# B&R Automation Studio project vibratorControlWithCurrentController (part 7)

#### Variables.var - Local variables
```iecst
VAR CONSTANT
	CYCLE_TIME_us : REAL := 1600.0;
	CYCLE_TIME_s : REAL := 0.0016;
	PI : REAL := 3.1415926536;
END_VAR
VAR
	acc : acc_typ;
	i : USINT;
	vibratorControl_0 : ARRAY[0..NUM_VIBRATOR] OF vibratorControl := [2((startPercentBoost:=5))];
	local : ARRAY[0..NUM_VIBRATOR] OF local_typ;
	MTFilterMovingAverage_0 : ARRAY[0..NUM_VIBRATOR] OF MTFilterMovingAverage;
	MTBasicsTimeDelay_0 : ARRAY[0..NUM_VIBRATOR] OF MTBasicsTimeDelay;
	GetPhaseDifference_0 : ARRAY[0..NUM_VIBRATOR] OF GetPhaseDifference;
	hmiAccelerometerPercent : REAL;
END_VAR
```

#### LocalFunctions.fun
```iecst
{REDUND_ERROR} FUNCTION_BLOCK vibratorControl (*TODO: Add your comment here*) (*$GROUP=User,$CAT=User,$GROUPICON=User.png,$CATICON=User.png*)
	VAR_INPUT
		enable : BOOL;
		amplitude : REAL;
		percent : REAL;
		vibratorType : USINT;
		machineType : USINT;
		manualFrequency : REAL;
		manualControl : BOOL;
		linearizationAmplitude : ARRAY[0..4] OF REAL;
		linearizationFrequencies : ARRAY[0..4] OF REAL;
		pAxis : UDINT;
		manualBrake : BOOL;
		boostVelocityLow : REAL := 180;
		boostVelocityHigh : REAL;
		brakeVelocity : REAL;
		boostFrequency : REAL;
		brakeFrequency : REAL;
		boostAmplitude : REAL;
		brakeAmplitude : REAL;
		manualBoost : BOOL;
		currAccelerometerValue : REAL;
		currAccelerometerPercent : REAL;
		manualBrakeTime : REAL;
		manualBrakeAmplitudeEnd : REAL;
		manualBrakeFrequencyEnd : REAL;
		activateMinMax : BOOL;
		disableBoost : BOOL;
	END_VAR
	VAR_OUTPUT
		frequency_out : REAL;
		amplitude_out : REAL;
		phaseShift : REAL := 0;
		sin_out : REAL;
		accelerationStart : REAL;
		minAcceleration : REAL;
		minAccelerationTime : REAL;
		caliBoostVelocityLow : REAL;
		caliBoostVelocityHigh : REAL;
		estimatedPercent : REAL;
		minBreakPercent : REAL;
		maxBoostPercent : REAL;
		filteredAccelerometerPercent : REAL;
	END_VAR
	VAR
		state : UINT;
		oldPercent : REAL;
		phi : REAL;
		sine : REAL;
		time : REAL;
		oldMachineType : USINT := 222; (*222 to make sure gets initialized*)
		addBrakeAmplitude : REAL;
		enableBrake : BOOL := TRUE;
		phaseShiftLocal : REAL;
		minBrakeTime : REAL := 0;
		j : UINT;
		MTLookUpTable_0 : MTLookUpTable;
		frequency : REAL;
		MC_BR_CyclicWrite_0 : MC_BR_CyclicWrite;
		old_sin : REAL;
		sin_ref : REAL;
		startPercentBoost : REAL;
		sin_abs : REAL;
		oldVibratorType : USINT;
		brakeStartDelay : REAL;
		brakePercent : REAL;
		timeStart : REAL;
		accelerationStart20pct : REAL;
		MTDataMinMax_0 : MTDataMinMax;
		MTFilterMovingAverage_0 : MTFilterMovingAverage;
		oldCurrAccelerometerValue : REAL;
		boostHighLowSeperatorPercent : REAL := 50.0;
	END_VAR
END_FUNCTION_BLOCK

FUNCTION getPercentFromAcceleration : REAL
	VAR_INPUT
		acc : REAL;
		vibratorType : USINT; (*0=CF, 1=LF*)
		machineType : USINT; (*0=small, 1=big*)
	END_VAR
END_FUNCTION

FUNCTION getAccelerationFromPercent : REAL
	VAR_INPUT
		percent : REAL;
		vibratorType : USINT; (*0=CF, 1=LF*)
		machineType : USINT; (*0=small, 1=big*)
	END_VAR
END_FUNCTION

FUNCTION applyBrake : REAL
	VAR_INPUT
		percent : REAL;
		brakeVelocity : REAL; (*accValue/s*)
		vibratorType : USINT; (*0=CF, 1=LF*)
		machineType : USINT; (*0=small, 1=big*)
	END_VAR
	VAR
		acc : REAL;
		bigBowlChange : REAL := 48000;
	END_VAR
END_FUNCTION

FUNCTION applyBoost : REAL
	VAR_INPUT
		percent : REAL;
		boostVelocity : REAL; (*accValue/s*)
		vibratorType : USINT; (*0=CF, 1=LF*)
		machineType : USINT; (*0=small, 1=big*)
	END_VAR
	VAR
		acc : REAL;
	END_VAR
END_FUNCTION

FUNCTION_BLOCK GetPhaseDifference
	VAR_INPUT
		Enable : BOOL;
		ReferenceSignal : REAL;
		Signal : REAL;
	END_VAR
	VAR_OUTPUT
		Phase : REAL;
		PhaseInv : REAL;
	END_VAR
	VAR
		x : ARRAY[0..MAX_SIGNAL_LENGTH] OF REAL;
		y : ARRAY[0..MAX_SIGNAL_LENGTH] OF REAL;
		r : ARRAY[0..MAX_OUTPUT_LENGTH] OF REAL;
	END_VAR
	VAR CONSTANT
		MAX_SIGNAL_LENGTH : UINT := 19;
		MAX_OUTPUT_LENGTH : UINT := (MAX_SIGNAL_LENGTH*2)+1;
	END_VAR
	VAR
		i : {REDUND_UNREPLICABLE} UINT;
		sum : {REDUND_UNREPLICABLE} REAL;
		offset : {REDUND_UNREPLICABLE} INT;
		j : {REDUND_UNREPLICABLE} UINT;
		maxVal : {REDUND_UNREPLICABLE} REAL;
		maxIdx : {REDUND_UNREPLICABLE} UINT;
		state : UINT;
		idx : UINT;
		minVal : REAL;
		minIdx : UINT;
	END_VAR
END_FUNCTION_BLOCK
```

#### LocalFunctions.st
```iecst
FUNCTION_BLOCK vibratorControl

	CASE state OF

		0:
			IF enable THEN
				IF vibratorType=0 THEN
					state := 5;
				ELSE
					//LF
					state := 8;
				END_IF
			END_IF

		5: // CF Running
			IF manualControl THEN
				state := 200;
			ELSIF percent < estimatedPercent AND frequency <> 0.0 THEN
				time := 0;
				brakePercent := percent;
				state := 20;
			ELSIF percent > estimatedPercent AND frequency <> 0.0 THEN
				time := 0;
				oldPercent := percent;
				state := 10;
			ELSE
				amplitude_out := amplitude;
				MTLookUpTable_0.InX := amplitude;
				MTLookUpTable_0();
				frequency := MTLookUpTable_0.Out;
			END_IF

		8: // LF Running
			IF manualControl THEN
				state := 200;
			ELSE
				amplitude_out := amplitude;
				MTLookUpTable_0.InX := amplitude;
				MTLookUpTable_0();
				frequency := MTLookUpTable_0.Out;
			END_IF

		10: // wait for zero crossing
			IF sin_ref >= 0.0 AND old_sin < 0.0 THEN
				amplitude_out := boostAmplitude;
				estimatedPercent := MAX(estimatedPercent, startPercentBoost);

				MTDataMinMax_0.Enable := FALSE;
				MTDataMinMax_0();
				state := 15;
			ELSIF sin_ref <= 0.0 AND old_sin > 0.0 THEN
				amplitude_out := boostAmplitude;
				estimatedPercent := MAX(estimatedPercent, startPercentBoost);

				MTDataMinMax_0.Enable := FALSE;
				MTDataMinMax_0();
				state := 15;
			END_IF

		15: // Boosting
			amplitude_out := boostAmplitude;
			frequency := boostFrequency;

			IF estimatedPercent <= boostHighLowSeperatorPercent THEN
				estimatedPercent := applyBoost(estimatedPercent, boostVelocityLow, vibratorType, machineType);
			ELSE
				estimatedPercent := applyBoost(estimatedPercent, boostVelocityHigh, vibratorType, machineType);
			END_IF
			time := time + CYCLE_TIME_s;

			IF percent <> oldPercent THEN
				state := 5;
			ELSIF estimatedPercent >= percent OR disableBoost THEN
				estimatedPercent := percent;
				state := 5;
			END_IF

		20:
			IF sin_ref >= 0.0 AND old_sin < 0.0 THEN
				amplitude_out := brakeAmplitude;
				phi := phi - (PI/2.0);

				MTDataMinMax_0.Enable := FALSE;
				MTDataMinMax_0();
				state := 25;
			ELSIF sin_ref <= 0.0 AND old_sin > 0.0 THEN
				amplitude_out := brakeAmplitude;
				phi := phi - (PI/2.0);

				MTDataMinMax_0.Enable := FALSE;
				MTDataMinMax_0();
				state := 25;
			END_IF

		25: // Braking
			amplitude_out := brakeAmplitude;
			frequency := brakeFrequency;

			estimatedPercent := applyBrake(estimatedPercent, brakeVelocity, vibratorType, machineType);

			time := time + CYCLE_TIME_s;

			IF estimatedPercent <= brakePercent THEN
				estimatedPercent := brakePercent;

				amplitude_out := 0.0;
				phi := phi + (PI/2.0);
				state := 5;
			END_IF

		100:
			amplitude_out := amplitude;
			MTLookUpTable_0.InX := amplitude;
			MTLookUpTable_0();
			frequency := MTLookUpTable_0.Out;

		200:
			frequency := manualFrequency;
			amplitude_out := amplitude;

			IF manualBrake THEN
				state := 210;
				time := 0;
			ELSIF manualBoost THEN
				time := 0.0;
				state := 250;
			ELSIF NOT manualControl THEN
				estimatedPercent := 0;
				MTLookUpTable_0.Enable := FALSE;
				MTLookUpTable_0();
				state := 5;
			END_IF

		210:
			IF sin_ref >= 0.0 AND old_sin < 0.0 THEN
				amplitude_out := brakeAmplitude;
				phi := phi - (PI/2.0);
				accelerationStart := currAccelerometerValue;
				minAcceleration := 99999999;
				state := 220;
			ELSIF sin_ref <= 0.0 AND old_sin > 0.0 THEN
				amplitude_out := brakeAmplitude;
				phi := phi - (PI/2.0);
				accelerationStart := currAccelerometerValue;
				timeStart := 0;
				minAcceleration := 99999999;
				state := 220;
			END_IF

		220: // Braking
			amplitude_out := brakeAmplitude;
			frequency := brakeFrequency;

			time := time + CYCLE_TIME_s;

			IF time > manualBrakeTime OR NOT manualBrake THEN
				amplitude_out := manualBrakeAmplitudeEnd;
				frequency := manualBrakeFrequencyEnd;
				phi := phi + (PI/2.0);
				state := 230;
			END_IF

			IF currAccelerometerValue < minAcceleration THEN
				IF timeStart > 0 AND time-timeStart >= CYCLE_TIME_s*2 THEN
					accelerationStart := accelerationStart20pct;
					minAcceleration := currAccelerometerValue;
					minAccelerationTime := time-timeStart;
				ELSE
					minAcceleration := currAccelerometerValue;
					minAccelerationTime := time;
				END_IF
			END_IF

			// If acceleromter falls more than 20% save that point as "start point".
			IF currAccelerometerValue < (accelerationStart*0.8) AND timeStart=0 THEN
				accelerationStart20pct := currAccelerometerValue;
				timeStart := time;
			END_IF

		230:
			IF currAccelerometerValue < minAcceleration THEN
				IF timeStart > 0 AND time-timeStart >= CYCLE_TIME_s*2 THEN
					accelerationStart := accelerationStart20pct;
					minAcceleration := currAccelerometerValue;
					minAccelerationTime := time-timeStart;
				ELSE
					minAcceleration := currAccelerometerValue;
					minAccelerationTime := time;
				END_IF
			END_IF

			// If acceleromter falls more than 20% save that point as "start point".
			IF currAccelerometerValue < (accelerationStart*0.8) AND timeStart=0 THEN
				accelerationStart20pct := currAccelerometerValue;
				timeStart := time;
			END_IF

			IF NOT manualBrake THEN
				amplitude_out := 0;
				state := 200;
			END_IF

		250: // wait for zero crossing
			IF sin_ref >= 0.0 AND old_sin < 0.0 THEN
				amplitude_out := boostAmplitude;
				state := 260;
			ELSIF sin_ref <= 0.0 AND old_sin > 0.0 THEN
				amplitude_out := boostAmplitude;
				state := 260;
			END_IF

		260: // Boosting
			amplitude_out := boostAmplitude;
			frequency := boostFrequency;

			time := time + CYCLE_TIME_s;
			caliBoostVelocityLow := currAccelerometerValue / time;

			IF time >= 0.5 OR NOT manualBoost OR currAccelerometerPercent >= 50.0 THEN
				time := 0;
				accelerationStart := currAccelerometerValue;
				state := 270;
			END_IF

		270:
			amplitude_out := boostAmplitude;
			frequency := boostFrequency;

			time := time + CYCLE_TIME_s;
			caliBoostVelocityHigh := (currAccelerometerValue-accelerationStart) / time;

			IF time >= 0.5 THEN
				caliBoostVelocityHigh := caliBoostVelocityLow;

				amplitude_out := 0.0;
				state := 280;
			ELSIF NOT manualBoost OR currAccelerometerPercent >= 90.0 THEN
				amplitude_out := 0.0;
				state := 280;
			END_IF

		280:
			IF NOT manualBoost THEN
				state := 200;
			END_IF

	END_CASE

	IF NOT enable AND state <> 0 THEN
		estimatedPercent := 0;
		state := 0;
		amplitude_out := 0;
		frequency_out := 0;
	END_IF

	// Lookup table for frequencies
	IF enable AND NOT MTLookUpTable_0.Enable THEN
		MTLookUpTable_0.Mode := mtLOOKUP_LINEAR_EXTRAPOLATION;

		MTLookUpTable_0.NumberOfNodes := 0;
		FOR j:=0 TO 4 DO
			IF linearizationAmplitude[j]=0.0 THEN
				EXIT;
			END_IF
			MTLookUpTable_0.NodeVectorX[j] := linearizationAmplitude[j];
			MTLookUpTable_0.FcnValues[j] := linearizationFrequencies[j];
			MTLookUpTable_0.NumberOfNodes := MTLookUpTable_0.NumberOfNodes + 1;
		END_FOR
	END_IF
	MTLookUpTable_0.Enable := enable;
	MTLookUpTable_0();

	IF activateMinMax OR manualControl THEN
		IF currAccelerometerValue <> oldCurrAccelerometerValue THEN
			oldCurrAccelerometerValue := currAccelerometerValue;

			MTFilterMovingAverage_0.Enable := TRUE;
			MTFilterMovingAverage_0.In := currAccelerometerValue;
			MTFilterMovingAverage_0.WindowLength := 10;
			MTFilterMovingAverage_0();

			MTDataMinMax_0.Enable := TRUE;
			MTDataMinMax_0.In := MTFilterMovingAverage_0.Out;
			MTDataMinMax_0();
			minBreakPercent := getPercentFromAcceleration(MTDataMinMax_0.MinValue ,vibratorType,machineType);
			maxBoostPercent := getPercentFromAcceleration(MTDataMinMax_0.MaxValue ,vibratorType,machineType);
			filteredAccelerometerPercent := getPercentFromAcceleration(MTFilterMovingAverage_0.Out,vibratorType,machineType);
		END_IF
	END_IF

	old_sin := sin_ref;

	// create sinewave amplitude with defined frequency
	sin_out := amplitude_out*SIN(phi+phaseShift);
	sin_abs := ABS(sin_out);
	phi := fmod(phi + frequency*2*PI*CYCLE_TIME_s, 2*PI);
	sin_ref := SIN(phi+phaseShift);
	phaseShift := fmod(phaseShift, 2*PI);
	phaseShiftLocal := fmod(phaseShiftLocal, 2*PI);

	// Write sine wave to vibrator parID
	MC_BR_CyclicWrite_0.Enable := enable;
	MC_BR_CyclicWrite_0.Axis := pAxis;
	MC_BR_CyclicWrite_0.DataType := ncPAR_TYP_REAL;
	MC_BR_CyclicWrite_0.DataAddress := ADR(sin_out);
	MC_BR_CyclicWrite_0.ParID := ACP10PAR_USER_R4_VAR1;
	MC_BR_CyclicWrite_0();

	// If machineType changes we must change parameters.
	IF machineType <> oldMachineType OR vibratorType <> oldVibratorType THEN
		oldMachineType := machineType;
		oldVibratorType := vibratorType;

		IF machineType=0 THEN
			IF vibratorType=0 THEN
				// small CF
			//	startPercentBoost := 5.0;
				brakeAmplitude := 1.5;
				boostAmplitude := 1.5;
				boostVelocityLow := 60500;
			ELSE
				// small LF
			//	startPercentBoost := 10.0;
				brakeAmplitude := 0.06;
				boostAmplitude := 0.12;
				boostVelocityLow := 29195;
			END_IF
		ELSE
			IF vibratorType=0 THEN
				// big CF
			//	startPercentBoost := 5.0;
				brakeAmplitude := 2.5;
				boostAmplitude := 2.5;
				boostVelocityLow := 29195;
			ELSE
				// big LF
			//	startPercentBoost := 10.0;
				brakeAmplitude := 0.06;
				boostAmplitude := 0.12;
				boostVelocityLow := 29195;
			END_IF
		END_IF

	END_IF

END_FUNCTION_BLOCK

FUNCTION getPercentFromAcceleration

	IF machineType=0 THEN
		IF vibratorType=0 THEN
			// 10%=2756 , 100%=17420
			getPercentFromAcceleration := (acc-1126.7)/162.93;
		ELSE
			// 10%=1300 , 100%=10140
			getPercentFromAcceleration := (acc-317.78)/98.222;
		END_IF
	ELSE
		IF vibratorType=0 THEN
			// 10%=1456 , 100%=8060
			getPercentFromAcceleration := (acc-722.22)/73.378;;
		ELSE
			// 10%=1508 , 100%=8840
			getPercentFromAcceleration := (acc-693.33)/81.467;
		END_IF
	END_IF

END_FUNCTION

FUNCTION getAccelerationFromPercent

	IF machineType=0 THEN
		IF vibratorType=0 THEN
			// 10%=2756 , 100%=17420
			getAccelerationFromPercent := percent*162.93+1126.7;
		ELSE
			// 10%=1300 , 100%=10140
			getAccelerationFromPercent := percent*98.222+317.78;
		END_IF
	ELSE
		IF vibratorType=0 THEN
			// 10%=1456 , 100%=8060
			getAccelerationFromPercent := percent*73.378+722.22;
		ELSE
			// 10%=1508 , 100%=8840
			getAccelerationFromPercent := percent*81.467+693.33;
		END_IF
	END_IF

END_FUNCTION

FUNCTION applyBoost
	acc := getAccelerationFromPercent(percent,vibratorType,machineType);
	applyBoost := getPercentFromAcceleration(acc+(boostVelocity*CYCLE_TIME_s),vibratorType,machineType);

//	IF machineType=0 THEN
//		IF vibratorType=0 THEN
//			applyBoost := getPercentFromAcceleration(acc+(55910*CYCLE_TIME_s),vibratorType,machineType);
//		ELSE
//			applyBoost := getPercentFromAcceleration(acc+(29195*CYCLE_TIME_s),vibratorType,machineType);
//		END_IF
//	ELSE
//		IF vibratorType=0 THEN
//			// big CF
//			applyBoost := getPercentFromAcceleration(acc+(29195*CYCLE_TIME_s),vibratorType,machineType);
//		ELSE
//			applyBoost := getPercentFromAcceleration(acc+(29195*CYCLE_TIME_s),vibratorType,machineType);
//		END_IF
//	END_IF

END_FUNCTION

FUNCTION applyBrake
	acc := getAccelerationFromPercent(percent,vibratorType,machineType);
	applyBrake := getPercentFromAcceleration(acc-(brakeVelocity*CYCLE_TIME_s),vibratorType,machineType);

	//	IF vibratorSize=0 THEN
	//		IF vibratorType=0 THEN
	//			applyBrake := getPercentFromAcceleration(acc-(48000*CYCLE_TIME_s),vibratorType,vibratorSize); //applyBrake := getPercentFromAcceleration(acc-(94349*CYCLE_TIME_s),vibratorType,vibratorSize);
	//		ELSE
	//			applyBrake := getPercentFromAcceleration(acc-(48000*CYCLE_TIME_s),vibratorType,vibratorSize);
	//		END_IF
	//	ELSE
	//		IF vibratorType=0 THEN
	//			// big CF
	//			applyBrake := getPercentFromAcceleration(acc-(42000*CYCLE_TIME_s),vibratorType,vibratorSize);
	//		ELSE
	//			applyBrake := getPercentFromAcceleration(acc-(48000*CYCLE_TIME_s),vibratorType,vibratorSize);
	//		END_IF
	//	END_IF

END_FUNCTION

FUNCTION_BLOCK GetPhaseDifference

	CASE state OF
		0:
			IF Enable THEN
				idx := 0;
				state := 10;
			END_IF

		10:
			x[idx] := ReferenceSignal;
			y[idx] := Signal;

			idx := idx + 1;

			IF idx > MAX_SIGNAL_LENGTH THEN
				idx := 0;
				state := 20;
			END_IF

		20:
			maxVal := 0;
			maxIdx := 0;
			minVal := 999999999;
			minIdx := 0;

			FOR i:=0 TO MAX_OUTPUT_LENGTH DO
				sum := 0;
				offset := UINT_TO_INT(i)-UINT_TO_INT(MAX_SIGNAL_LENGTH);
				FOR j:=0 TO MAX_SIGNAL_LENGTH DO
					IF UINT_TO_INT(j)+offset >= 0 AND UINT_TO_INT(j)+offset <= MAX_SIGNAL_LENGTH THEN
						sum := sum + (x[j] * y[j+offset]);
					END_IF
				END_FOR
				IF sum >= maxVal THEN
					maxVal := sum;
					maxIdx := i;
				END_IF
				IF sum <= minVal THEN
					minVal := sum;
					minIdx := i;
				END_IF

				r[i] := sum;
			END_FOR

			Phase := UINT_TO_REAL(maxIdx)-UINT_TO_REAL(MAX_SIGNAL_LENGTH);
			PhaseInv := UINT_TO_REAL(minIdx)-UINT_TO_REAL(MAX_SIGNAL_LENGTH);

			state := 10;

	END_CASE

	IF NOT Enable AND state > 0 THEN
		state := 0;
	END_IF

END_FUNCTION_BLOCK
```

### Program Logical/modules/main/vibrator/VibratorControl (IEC)

#### local.st - Init, cyclic, exit code
```iecst
PROGRAM _INIT

	FOR i:=0 TO NUM_VIBRATOR DO
		this ACCESS ADR(localVariables[i]);
		config ACCESS ADR(localVariables[i].config);

		// gets the task name and setup names for config and receipe types
		ST_name(0,ADR(this.configName),0);
		brdkStrCat(ADR(this.configName),ADR(':localVariables['));
		brdkStrAppendUdintToA(i,ADR(this.configName),0,-1);
		brdkStrCat(ADR(this.configName),ADR('].config'));

		this.VibFeedback_0.VibratorType := i;
		this.VibControl_0.VibratorType := i; // i=0=CF , i=1=LF
		this.Accelerometer_0.VibratorType := i; // i=0=CF , i=1=LF
		this.MpRecipeRegPar_Config.Enable := TRUE;
		config.emptyPercent := SEL(i=0,110,50);
		gVibratorInterface[i].cmd.emptyPercent := config.emptyPercent;
	END_FOR

END_PROGRAM

PROGRAM _CYCLIC

	FOR i:=0 TO NUM_VIBRATOR DO
		this ACCESS ADR(localVariables[i]);
		config ACCESS ADR(localVariables[i].config);
		hmi ACCESS ADR(localHmi[i]);

		modules;
	END_FOR

	// Watch Idx
	i := LIMIT(0, watchIdx, NUM_VIBRATOR);
	this ACCESS ADR(localVariables[i]);
	hmi ACCESS ADR(localHmi[i]);
	config ACCESS ADR(localVariables[i].config);

END_PROGRAM

PROGRAM _EXIT

END_PROGRAM
```

#### modules.st
```iecst
ACTION modules:

	// Function block for accelerometer processing
	this.Accelerometer_0.Enable := this.Accelerometer_0.ModuleOkCalibrationTool OR this.Accelerometer_0.ModuleOkBusCtrl;
	this.Accelerometer_0();

	// Function block for calculating airgap phase and amplitude
	this.VibFeedback_0.Enable := gVibratorInterface[i].status.powered;
	this.VibFeedback_0.Axis := SEL(i=0, ADR(gAxisVibL), ADR(gAxisVibC));
	this.VibFeedback_0.Amplitude_out := this.VibControl_0.amplitude_out;
	this.VibFeedback_0.Frequency := this.VibControl_0.frequency_out;
	this.VibFeedback_0.HoldPhase := this.VibControl_0.HoldPhase;
	this.VibFeedback_0.SinePhase := this.VibControl_0.SinePhase;
	this.VibFeedback_0.SineOut := this.VibControl_0.SineOut;
	this.VibFeedback_0.Braking := this.VibControl_0.Braking;
	this.VibFeedback_0.RawVib := this.Accelerometer_0.Raw; // only for phase verification
	this.VibFeedback_0.BrakingToAmplitudePct := this.VibControl_0.BrakingToAmplitudePct;
	this.VibFeedback_0();

	// Function block for closed loop phase and amplitude control, as well as setpoint generation for current controller
	this.VibControl_0.Enable := gVibratorInterface[i].status.powered;
	this.VibControl_0.Axis := SEL(i=0, ADR(gAxisVibL), ADR(gAxisVibC));
	this.VibControl_0.Percent := this.Accelerometer_0.Percent;
	this.VibControl_0.SetAmplitude := gVibratorInterface[i].status.percent;
	this.VibControl_0.ActPhase := this.VibFeedback_0.Phase;
	this.VibControl_0.ActPhaseValid := this.VibFeedback_0.PhaseValid;
	this.VibControl_0.ActPhaseAcc := this.VibFeedback_0.PhaseAcc;
	this.VibControl_0.ActAmplitude := SEL(this.testAccFeedback,this.VibFeedback_0.Amplitude,this.Accelerometer_0.Percent);
	this.VibControl_0.ActAmplitudeValid := this.VibFeedback_0.AmplitudeValid;
	this.VibControl_0.ManualControl := (gVibratorInterface[i].status.forcing) AND NOT gVibratorInterface[i].status.caliProdTest;
//	this.VibControl_0.AccPercent := this.Accelerometer_0.Percent;
	this.VibControl_0();
	hmi.frequencyTimes2 := this.VibControl_0.frequency_out*2.0; // to show on HMI

	// Config handling (it takes too much CPU to run in 0.8ms so we run it with a timer):
	this.timeConfig := this.timeConfig + CYCLE_TIME_us;
	IF this.timeConfig > 80000 THEN // 80ms
		this.timeConfig := 0;

		// Slow inputs every 80ms
		this.VibControl_0.config := ADR(config);
		this.VibFeedback_0.config := ADR(config);
		this.VibFeedback_0.UpdateFilter := this.VibControl_0.UpdateFilter;
		this.VibFeedback_0.Calibrating := gVibratorInterface[i].status.calibratingMode AND NOT this.VibControl_0.TestPulses;
		this.Accelerometer_0.MachineSize := config.MachineSize;
		this.VibFeedback_0.MachineSize := config.MachineSize;
		this.VibControl_0.MachineSize := config.MachineSize;
		this.VibControl_0.Calibrate := gVibratorInterface[i].status.calibratingMode;
		this.VibControl_0.RampUp := SEL(gVibratorInterface[i].status.rampUp > 0,0,100/(INT_TO_REAL(gVibratorInterface[i].status.rampUp)/1000)); // ms it takes to go from 0% to 100% -> 100ms ex. 100/0.1 = 1000%/s
		this.VibControl_0.ManualPercent := SEL(gVibratorInterface[i].parameter.speedPctManualTest > 0,this.VibControl_0.ManualPercent,gVibratorInterface[i].parameter.speedPctManualTest);
		this.VibControl_0.MinTimeInCount := config.minTimeInCount;
		this.VibControl_0.MinTimeInCountBigCf := config.minTimeInCountBigCf;

		// Slow outputs every 80ms
		gVibratorInterface[i].cmd.calibrationDone := this.VibControl_0.CalibrateDone;
		gVibratorInterface[i].cmd.testPulses := this.VibControl_0.TestPulses;
		gVibratorInterface[i].cmd.emptyPercent := config.emptyPercent;
		gVibratorInterface[i].parameter.machineSize := localVariables[0].config.MachineSize;
		this.VibControl_0.UpdateFilterDone := this.VibFeedback_0.UpdateFilterDone;
		localVariables[1].config.MachineSize := localVariables[0].config.MachineSize;
		hmi.calibrationNotActive := NOT this.VibControl_0.Calibrate;

		IF config.calibrationDone THEN
			config.timeInCalibrationSeconds := config.timeInCalibrationSeconds + 0.08; // Previously used PLC TIME but that gets destroyed by NTP. Rather use a counter even though it can't count if power is OFF.
			hmi.daysSinceCalibration := config.timeInCalibrationSeconds/86400; // Convert seconds to days.

			// Auto save every 30min
			timeElapsedMillis := timeElapsedMillis + 80;
			IF timeElapsedMillis > 1800000 THEN
				timeElapsedMillis := 0;
				this.SaveConfig := TRUE;
			END_IF

			// Only show this when calibration is done. Otherwise it will show 2 different numbers doing calibration which may confuse
			config.ressonanceFrequencyAt45Pct := config.maxFrequencySweep*2.0; // ressonance (mechanical) frequency is really 2 times output frequency.
		ELSE
			hmi.daysSinceCalibration := 99999;
		END_IF

		// Set max current depending which machine size.
		IF config.MachineSize=0 THEN
			this.VibControl_0.MaxCurr := SEL(i=0, 0.20, 2.0);
		ELSE
			this.VibControl_0.MaxCurr := SEL(i=0, 0.20, 3.1);
		END_IF

		// Set max current depending which machine size.
		IF config.MachineSize=0 THEN
			// Small bowl						  LF    CF
			hmi.minResonanceFrequency := SEL(i=0, 96, 96);
			hmi.maxResonanceFrequency := SEL(i=0, 106, 102);
			hmi.minCurrent := SEL(i=0, 0.04, 0.4);
			hmi.maxCurrent := SEL(i=0, 0.13, 1.3);
		ELSE
			// Big bowl							  LF    CF
			hmi.minResonanceFrequency := SEL(i=0, 96, 47);
			hmi.maxResonanceFrequency := SEL(i=0, 106, 52);
			hmi.minCurrent := SEL(i=0, 0.04, 0.4);
			hmi.maxCurrent := SEL(i=0, 0.13, 1.9);
		END_IF
		hmi.resonanceFrequencyOK := this.config.ressonanceFrequencyAt45Pct >= hmi.minResonanceFrequency AND this.config.ressonanceFrequencyAt45Pct <= hmi.maxResonanceFrequency;
		hmi.currentOK := this.config.maxCurrentUsed >= hmi.minCurrent AND this.config.maxCurrentUsed <= hmi.maxCurrent;

		// Interface calibration results to FAT (send if calibrate is stopped)
		IF this.VibControl_0.SendCaliResultToFAT THEN
			this.VibControl_0.SendCaliResultToFAT := FALSE;

			gVibratorInterface[i].status.calibrationResultFrequencyOK := hmi.resonanceFrequencyOK;
			gVibratorInterface[i].status.calibrationResultCurrentOK := hmi.currentOK;
			gVibratorInterface[i].status.calibrationResultFrequency := this.config.ressonanceFrequencyAt45Pct;
			gVibratorInterface[i].status.calibrationResultCurrent := this.config.maxCurrentUsed;
			gVibratorInterface[i].status.calibrationResultsReady := TRUE;
		END_IF
		gVibratorInterface[i].status.calibrationDone := config.calibrationDone;

		// set machinesize (cmd from FAT)
		IF gVibratorInterface[i].cmd.setCfType THEN
			gVibratorInterface[i].cmd.setCfType := FALSE;
			config.MachineSize := gVibratorInterface[i].parameter.CFType; //0=small , 1=big
			this.SaveConfig := TRUE;
		END_IF

		// State Machine to save config.
		CASE this.stateSave OF

			0:
				IF this.VibControl_0.SaveConfig AND gConfig.status.loaded THEN
					// Save from calibration
					gConfig.cmd.save := TRUE;
					gMachineInterface.cmd.requestSaveToT50 := TRUE;
					this.stateSave := 10;
				ELSIF this.SaveConfig AND gConfig.status.loaded THEN
					// Save because HMI variable changed.
					this.SaveConfig := FALSE;
					gConfig.cmd.save := TRUE;
					this.stateSave := 30;
				END_IF

			10:
				IF NOT gConfig.cmd.save THEN
					this.VibControl_0.SaveConfigDone := TRUE;
					this.stateSave := 20;
				END_IF

			20:
				IF NOT this.VibControl_0.SaveConfig THEN
					this.VibControl_0.SaveConfigDone := FALSE;
					this.stateSave := 0;
				END_IF

			30:
				IF NOT gConfig.cmd.save THEN
					this.stateSave := 0;
				END_IF

		END_CASE

	this.MpRecipeRegPar_Config(MpLink := ADR(mpRecipe), PVName := ADR(this.configName), Category := ADR('config'));
END_IF

END_ACTION
```

#### Types.typ - Local data types
```iecst
TYPE
	hmi_typ : 	STRUCT
		NeedCalibration : BOOL;
		CalibrationStatus : calibrationResult_enum;
		daysSinceCalibration : REAL := 99999;
		calibrationNotActive : BOOL;
		resonanceFrequencyOK : BOOL;
		currentOK : BOOL;
		minCurrent : REAL;
		maxCurrent : REAL;
		minResonanceFrequency : REAL;
		maxResonanceFrequency : REAL;
		frequencyTimes2 : REAL;
	END_STRUCT;
	local_typ : 	STRUCT
		VibFeedback_0 : VibFeedback;
		VibControl_0 : VibControl;
		Accelerometer_0 : Accelerometer;
		useAccPhase : BOOL;
		MpRecipeRegPar_Config : MpRecipeRegPar;
		VibFeedback_old : VibFeedbackOld;
		configName : STRING[80];
		config : VibControl_config_typ;
		configOld : VibControl_config_typ;
		oldCheckChangesConfig : BOOL;
		timeConfig : UDINT;
		oldLoaded : BOOL;
		stateSave : USINT;
		testAccFeedback : BOOL;
		SaveConfig : BOOL;
	END_STRUCT;
	calibrationResult_enum :
		(
		CALIBRATION_NOT_DONE := 0,
		SMALL_CF_CALIBRATION_OK := 1,
		SMALL_CF_CALIBRATION_NOK := 2,
		BIG_CF_CALIBRATION_OK := 3,
		BIG_CF_CALIBRATION_NOK := 4,
		LF_CALIBRATION_OK := 5,
		LF_CALIBRATION_NOK := 6
		);
END_TYPE
```

#### Variables.var - Local variables
```iecst
VAR
	i : USINT;
END_VAR
VAR CONSTANT
	MAX_VIBRATORS : USINT := 1;
END_VAR
VAR
	localHmi : ARRAY[0..MAX_VIBRATORS] OF hmi_typ;
	localVariables : ARRAY[0..MAX_VIBRATORS] OF local_typ;
	this : REFERENCE TO local_typ;
	config : REFERENCE TO VibControl_config_typ;
	hmi : REFERENCE TO hmi_typ;
	watchIdx : USINT;
	timeElapsedMillis : UDINT;
END_VAR
```

#### LocalFunctions.fun
```iecst
{REDUND_ERROR} FUNCTION_BLOCK Accelerometer (*TODO: Add your comment here*) (*$GROUP=User,$CAT=User,$GROUPICON=User.png,$CATICON=User.png*)
	VAR_INPUT
		Enable : {REDUND_UNREPLICABLE} BOOL;
		VibratorType : USINT;
		MachineSize : USINT; (*0=Small CM, 1=Big CM*)
	END_VAR
	VAR_OUTPUT
		ModuleOkBusCtrl : BOOL; (*If using buscontroller*)
		ModuleOkCalibrationTool : BOOL;
		Percent : {REDUND_UNREPLICABLE} REAL;
		Raw : {REDUND_UNREPLICABLE} REAL;
		ai_rawValue : REAL;
		ai_peakValue : REAL;
		ai_rawValueBusCtrl : REAL;
		ai_peakValueBusCtrl : REAL;
		do_enableSampling : BOOL := TRUE;
		ao_samples : UINT := 103;
		isBigCF : BOOL;
	END_VAR
END_FUNCTION_BLOCK

FUNCTION CheckCalibrationFrequency : calibrationResult_enum
	VAR_INPUT
		ressFrequency : REAL;
		MachineSize : USINT;
		VibratorType : USINT;
	END_VAR
END_FUNCTION
```

#### LocalFunctions.st
```iecst
(* TODO: Add your comment here *)
FUNCTION_BLOCK Accelerometer

	IF Enable THEN
		IF ModuleOkBusCtrl THEN
			ai_peakValue := ai_peakValueBusCtrl;
			ai_rawValue := ai_rawValueBusCtrl;
			do_enableSampling := TRUE;
			ao_samples := SEL(MachineSize=1,53,103);		// Big bowl cf is half the frequency and need to use more samples in the accelerometer module.
		END_IF

		IF VibratorType=0 THEN
			Percent := SEL(MachineSize=0,(ai_peakValue-722.22)/73.378,(ai_peakValue-1300)/150);
		ELSE
			Percent := SEL(MachineSize=0,(ai_peakValue-693.33)/81.467,(ai_peakValue-317.78)/98.222); 			// 10%=1300 , 100%=10140
		END_IF
		Raw := ai_rawValue;
		isBigCF := MachineSize=1;
	ELSE
		Percent := 0.0;
		Raw := 0.0;
	END_IF

	// Small CF:		10%=2756 , 100%=17420
	// Small LF:		10%=1300 , 100%=10140
	// Big CF:			10%=1456 , 100%=8060
	// Big LF: 			10%=1508 , 100%=8840

END_FUNCTION_BLOCK

FUNCTION CheckCalibrationFrequency

	IF VibratorType=0 THEN
		//CF
		CASE MachineSize OF

			0:
				// small CF
				IF ressFrequency < 15 THEN
					CheckCalibrationFrequency := CALIBRATION_NOT_DONE;
				ELSIF ressFrequency < 96.0 OR ressFrequency > 102 THEN
					CheckCalibrationFrequency := SMALL_CF_CALIBRATION_NOK;
				ELSE
					CheckCalibrationFrequency := SMALL_CF_CALIBRATION_OK;
				END_IF

			1:
				// big CF
				IF ressFrequency < 15 THEN
					CheckCalibrationFrequency := CALIBRATION_NOT_DONE;
				ELSIF ressFrequency < 47.0 OR ressFrequency > 52.0 THEN
					CheckCalibrationFrequency := BIG_CF_CALIBRATION_NOK;
				ELSE
					CheckCalibrationFrequency := BIG_CF_CALIBRATION_OK;
				END_IF

		END_CASE

	ELSE
		//LF
		IF ressFrequency < 15 THEN
			CheckCalibrationFrequency := CALIBRATION_NOT_DONE;
		ELSIF ressFrequency < 96.0 OR ressFrequency > 106 THEN
			CheckCalibrationFrequency := LF_CALIBRATION_NOK;
		ELSE
			CheckCalibrationFrequency := LF_CALIBRATION_OK;
		END_IF
	END_IF

END_FUNCTION
```

### Library Logical/modules/main/vibrator/VibCtrl (IEC)

#### Types.typ - Exported data types
```iecst
TYPE
	lookup_typ : 	STRUCT
		key : REAL;
		value : REAL;
		error : REAL;
	END_STRUCT;
	VibControlCalibration_typ : 	STRUCT
		sweepAmplitude : REAL;
		sweepAmplitudeBigCF : REAL;
		MTDataStatistics_0 : MTDataStatistics;
		sweepTimeSteps : REAL := 0.3;
		sweepMaxAmplitude : REAL;
		sweepMaxFrequency : REAL;
		sweepMaxPhase : REAL;
		freqStepSize : REAL := 0.1;
		freqStepSizeSmall : REAL := 0.02;
		phaseStepSize : REAL := 2.50;
		stepTimeAmplitude : REAL := 4.0;
		startAmplitude : REAL := 0.3;
		stopAmplitude : REAL;
		stepSizeAmplitude : REAL := 0.1;
		setAmplitude : REAL;
		timePulseTest : REAL;
		bestTimePulseTest : REAL := 9999;
		startPulseTime : BOOL;
		saveMax : BOOL;
		sweepEndFrequency : REAL;
		countPulses : USINT;
		bestBoostCurrent : REAL;
	END_STRUCT;
	VibControl_config_typ : 	STRUCT
		MachineSize : USINT; (*0=Small CM, 1=Big CM*)
		lookUpPercentFromAmplitude : LUT_typ;
		lookUpCurrentFromPercent : LUT_typ;
		lookupFrequencyFromPercent : LUT_typ;
		lookupPhaseTargetFromPercent : LUT_typ;
		lookupFrequencyFromCurrent : LUT_typ;
		lookupBoostCurrentFromPercent : LUT_typ := (X:=[10,20,40,60,80,100,14(0.0)],Y:=[1.7,1.5,1.3,1.2,2(1.1),14(0.0)]);
		maxFrequencySweep : REAL;
		maxFrequencySweep2 : REAL;
		maxPhaseSweep : REAL;
		maxCurrentUsed : REAL;
		centerFrequencyBPF : REAL := 75.0;
		machineType : USINT; (*0=small bowl , 1=big bowl*)
		AddToBoostCurrentAt60pct : REAL; (*Current that was added to boost current at 60% (because we use 60% in calibration)*)
		boostCurrentScale : REAL := 1.4; (*Factor to scale ex. 0.10 which means that all boost currents will be scaled with +10% (could also be negative)*)
		OffsetBoostAmplitude : REAL;
		PhaseTarget : REAL := 70.0;
		emptyPercent : REAL;
		timeBoostCalibration : REAL;
		LUTsDescending : BOOL; (*TRUE if 1 or more LUTs are descending which is wrong!*)
		minTimeInCount : TIME := T#250ms;
		minTimeInCountBigCf : TIME := T#400ms;
		vibratorIsCalibrated : BOOL;
		ressonanceFrequencyAt45Pct : REAL; (*mechanical frequency = 2 * output frequnecy*)
		timeInCalibrationSeconds : REAL;
		calibrationDone : BOOL;
	END_STRUCT;
END_TYPE
```

#### Constants.var - Exported constants
```iecst
VAR CONSTANT
	VIB_CALI_PULSE_AMPLITUDE : REAL := 60.0;
	MAX_CALI_PULSES : USINT := 10;
	CYCLE_TIME_s : REAL := 0.0008;
	CYCLE_TIME_us : UDINT := 800;
	MAX_ELEMENTS : USINT := 5;
	MAX_LUT_IDX : USINT := 14;
	PI : REAL := 3.1415926536;
END_VAR
```

#### VibCtrl.fun - Exported functions and function blocks
```iecst
FUNCTION GetBrakeTimeFromAmplitude : REAL
	VAR_INPUT
		CurrentAmplitude : REAL;
		PercentChange : REAL;
		MachineSize : USINT;
	END_VAR
	VAR
		b : REAL := 40;
	END_VAR
END_FUNCTION

FUNCTION HammingWindow : REAL
	VAR_INPUT
		n : UINT;
		N : UINT;
	END_VAR
END_FUNCTION

FUNCTION GetPhaseTargetFromFrequency : REAL
	VAR_INPUT
		Frequency : REAL;
	END_VAR
END_FUNCTION

FUNCTION GetCurrentFromAmplitude : REAL
	VAR_INPUT
		Amplitude : REAL;
	END_VAR
END_FUNCTION

FUNCTION GetFrequencyFromAmplitude : REAL
	VAR_INPUT
		Amplitude : REAL;
	END_VAR
END_FUNCTION

FUNCTION GetPercentFromAmplitude : REAL
	VAR_INPUT
		Amplitude : REAL;
	END_VAR
END_FUNCTION

FUNCTION GetKpFromPercent : REAL
	VAR_INPUT
		Amplitude : REAL;
	END_VAR
END_FUNCTION

FUNCTION_BLOCK KalmanFilter1D
	VAR_INPUT
		Enable : BOOL;
		Measurement : REAL;
		KalmanGain : REAL;
		ProcessVariance : REAL;
		MeasureVariance : REAL;
	END_VAR
	VAR_OUTPUT
		Active : BOOL;
		Prediction : REAL;
		Estimation : REAL;
		ErrorEstimate : REAL;
	END_VAR
	VAR
		state : INT;
	END_VAR
END_FUNCTION_BLOCK

FUNCTION_BLOCK PIController
	VAR_INPUT
		Enable : BOOL;
		Hold : BOOL;
		LoopRate : TIME;
		Setpoint : REAL;
		ProcessValue : REAL;
		Kp : REAL;
		Ki : REAL;
		MinOutput : REAL;
		MaxOutput : REAL;
		Integral : REAL;
		Output : REAL;
		FeedForward : REAL;
	END_VAR
	VAR_OUTPUT
		Active : BOOL;
		Error : REAL;
	END_VAR
	VAR
		state : INT;
		TON_LoopRate : TON;
	END_VAR
END_FUNCTION_BLOCK

FUNCTION_BLOCK VibFeedbackOld
	VAR_INPUT
		Enable : BOOL;
		Axis : UDINT;
		RunCalculation : BOOL;
		Frequency : REAL;
		Simulation : BOOL;
		SimCurrent : REAL;
		AirgapScale : REAL := 1;
		PhaseOffset : REAL;
		HoldPhase : BOOL;
		current : ARRAY[0..2] OF REAL;
		voltage : ARRAY[0..2] OF REAL;
	END_VAR
	VAR_OUTPUT
		Amplitude : REAL;
		AmplitudeFast : REAL;
		Phase : REAL;
		PhaseFast : REAL;
		PhaseHMI : REAL;
	END_VAR
	VAR
		dt : REAL := 0.0004; (*400�s*)
		state : INT;
		currentLPF : ARRAY[0..2] OF REAL;
		voltageLPF : ARRAY[0..2] OF REAL;
		MC_BR_CyclicRead_0 : MC_BR_CyclicRead;
		MC_BR_CyclicRead_1 : MC_BR_CyclicRead;
		MC_BR_CyclicRead_2 : MC_BR_CyclicRead;
		MC_BR_CyclicRead_3 : MC_BR_CyclicRead;
		MC_BR_CyclicRead_4 : MC_BR_CyclicRead;
		MC_BR_CyclicRead_5 : MC_BR_CyclicRead;
		MC_BR_CyclicRead_6 : MC_BR_CyclicRead;
		MC_BR_CyclicRead_7 : MC_BR_CyclicRead;
		i : INT;
		MTFilterLowPass_2 : MTFilterLowPass;
		MTFilterLowPass_1 : MTFilterLowPass;
		MTFilterLowPass_0 : MTFilterLowPass;
		tmpTime : REAL := 0;
		lastTmpTime : REAL;
		zeroVolt : REAL := 0;
		intVolt : ARRAY[0..2] OF REAL := [3(0)];
		j : USINT;
		phaseFound : BOOL;
		intVoltBuffer : ARRAY[0..255] OF REAL;
		intCurrBuffer : ARRAY[0..255] OF REAL;
		currentLPFBuffer : ARRAY[0..255] OF REAL;
		intEMF : ARRAY[0..255] OF REAL; (*Integral of EMF*)
		intCurr : ARRAY[0..2] OF REAL := [3(0)];
		a : REAL := 0; (*voltage slope*)
		Offshift : USINT := 1; (*Offset for the airgap calculation*)
		lastidx : USINT := 0; (*index to count samples to loop for airgap calculation*)
		peakVib : REAL := 0; (*Peak vibration*)
		res : REAL := 4.2; (*Resistance*)
		lastTmpTimeMinusDt : REAL;
		tmpTimeAirgap : REAL;
		lastsumAirgap : REAL := 0;
		airgap : ARRAY[0..255] OF REAL := [256(0)];
		counter : UINT;
		MTFilterLowPass_Phase : MTFilterLowPass;
		MTFilterLowPass_Ampl : MTFilterLowPass;
		MC_BR_CyclicReadDataInfo_0 : MC_BR_CyclicReadDataInfo;
		airgap1 : REAL;
		airgap2 : REAL;
		tmpAirgapTrace : USINT;
		intCurr1 : REAL;
		intCurr2 : REAL;
		intVolt1 : REAL;
		intVolt2 : REAL;
		voltZeroOffset : REAL;
		currZeroOffset : REAL;
		phaseCalc : REAL;
		setPhase : REAL := 95;
		indexJ : USINT;
		CutOffFrequency : REAL := 150;
		windLenAmp : UINT := 2;
		windLenPhase : UINT := 2;
		MTFilterLowPass_Current : MTFilterLowPass;
		MTFilterLowPass_Frequency : MTFilterLowPass;
		xi : REAL;
		omega : REAL;
		alpha : REAL;
		simCurr10Prc : REAL := 0.4;
		simCurr100Prc : REAL := 1.1;
		simResonance : REAL := 49;
		simPrc : REAL;
		phaseRes : REAL;
		tmpAirgap : REAL;
		MTFilterBandPass_Airgap : MTFilterBandPass;
		MTFilterBandPass_Voltage3rd : MTFilterBandPass;
		windLenAirgap : UINT := 50;
		TimeDelay_0 : TimeDelay;
		TimeDelayVoltage : REAL;
		TON_RunDelay : TON;
		CalcDelay : TIME := T#0ms;
		RunDelay : TIME := T#50ms;
		TON_CalcDelay : TON;
		RawAirgap : BOOL := TRUE;
		meanAirgap : REAL := 3.2;
		KalmanFilter1D_Ampl : KalmanFilter1D;
		MTBasicsDT1_ActAmpl : MTBasicsDT1;
		MTFilterBandPass_AirgapFast : MTFilterBandPass;
		voltage3rdHarmonic : ARRAY[0..255] OF REAL;
		idx : USINT;
		peak3rdHarmonic : REAL;
	END_VAR
END_FUNCTION_BLOCK

FUNCTION_BLOCK VibFeedback
	VAR_INPUT
		Enable : BOOL;
		Axis : UDINT;
		VibratorType : USINT;
		Frequency : REAL;
		Amplitude_out : REAL := 0.0;
		HoldPhase : BOOL;
		Braking : BOOL := FALSE;
		BrakingToAmplitudePct : REAL; (*Amplitude that we are currently braking to "open loop".*)
		RawVib : REAL;
		PhaseOffset : REAL := -80;
		Calibrating : BOOL;
		config : REFERENCE TO VibControl_config_typ;
		SinePhase : REAL;
		SineOut : REAL;
		UpdateFilter : BOOL;
		MachineSize : USINT; (*0=Small CM, 1=Big CM*)
	END_VAR
	VAR_OUTPUT
		Amplitude : REAL;
		AmplitudeRaw : REAL;
		AmplitudeGoertzel : REAL;
		AmplitudeFast : REAL;
		Phase : REAL;
		PhaseAcc : REAL;
		PhaseGoertzel : REAL;
		current : ARRAY[0..2] OF REAL;
		voltage : ARRAY[0..2] OF REAL;
		AmplitudeValid : BOOL;
		PhaseValid : BOOL;
		UpdateFilterDone : BOOL;
		ActAmplitudeGoertzel : REAL;
	END_VAR
	VAR
		state : USINT;
		MTFilterBandPass_3rdHarmonic : MTFilterBandPass;
		LookupTbl_Percent : LookupTbl;
		MC_BR_CyclicRead_0 : MC_BR_CyclicRead := (ParID:=14433,DataType:=ncPAR_TYP_REAL);
		MC_BR_CyclicRead_1 : MC_BR_CyclicRead := (ParID:=14425,DataType:=ncPAR_TYP_REAL);
		MC_BR_CyclicRead_2 : MC_BR_CyclicRead := (ParID:=14435,DataType:=ncPAR_TYP_REAL);
		MC_BR_CyclicRead_3 : MC_BR_CyclicRead := (ParID:=14427,DataType:=ncPAR_TYP_REAL);
		i : USINT;
		time : REAL;
		peakVib : REAL;
		peakCurr : REAL;
		cnt : USINT;
		cntAcc : USINT;
		lastBPF : REAL;
		tmpTime : REAL;
		dt : REAL := 0.0004;
		tmpTimeAirgap : REAL;
		lastRawVib : REAL;
		CalcPhasePosAcc : BOOL;
		CalcPhaseNegAcc : BOOL;
		CalcPhasePos : BOOL;
		CalcPhaseNeg : BOOL;
		voltageZeroCrossing : BOOL;
		AmplitudeCurrent : REAL;
		Feedback : REAL;
		tmpTimeAcc : REAL;
		lastTmpTimeAcc : REAL;
		lastCurrAcc : REAL;
		hammingIdx : UINT;
		hammingLength : UINT := 50;
		tmpPhase : REAL;
		feedbackInterpolation : REAL;
		lastSinePhase : REAL;
		MTFilterLowPass_Phase : MTFilterLowPass;
		MTFilterLowPass_Amplitude : MTFilterLowPass;
		oldUpdateFilter : BOOL;
		testPhaseUsingAcc : BOOL;
		hammingWindow : ARRAY[0..MAX_SAMPLES_GOERTZEL] OF REAL;
		j : INT;
		goertzelCount : INT;
		samples : ARRAY[0..MAX_SAMPLES_GOERTZEL] OF REAL;
		samplesCurr : ARRAY[0..MAX_SAMPLES_GOERTZEL] OF REAL;
		goertzelMagPhase_0 : goertzelMagPhase;
		goertzelMagPhase_1 : goertzelMagPhase;
		goertzelMagPhase_2 : goertzelMagPhase;
		goertzelMagPhase_3 : goertzelMagPhase;
		phase : ARRAY[0..3] OF REAL;
		oldGoertzelPhaseStart : REAL;
		goertzelRef : REAL;
		goertzelSignal : REAL;
		goertzelPhase : REAL;
		goertzelScaling : REAL := 1;
		goertzelPhaseStart : REAL;
		goertzelPhaseComp : REAL;
		TON_PhaseValid : TON;
		timeHalfPeriod : REAL;
	END_VAR
END_FUNCTION_BLOCK

FUNCTION_BLOCK VibControl
	VAR_INPUT
		Enable : BOOL;
		Calibrate : BOOL;
		Percent : REAL;
		Axis : UDINT;
		ActPhase : REAL;
		ActPhaseAcc : REAL;
		SetAmplitude : REAL;
		ActAmplitude : REAL;
		ActAmplitudeValid : BOOL;
		ManualControl : BOOL;
		ManualCurrent : REAL;
		ManualPercent : REAL;
		ManualFrequency : REAL := 50.0;
		ClosedLoopAmplitude : BOOL;
		ClosedLoopPhase : BOOL;
		VibratorType : USINT;
		MaxCurr : REAL := 1.9;
		AccPercent : REAL;
		config : REFERENCE TO VibControl_config_typ;
		ActPhaseValid : BOOL;
		SaveConfigDone : BOOL;
		UpdateFilterDone : BOOL;
		MachineSize : USINT; (*0=Small CM, 1=Big CM*)
		MinTimeInCount : TIME := T#300ms;
		MinTimeInCountBigCf : TIME;
		RampUp : REAL; (*ms it takes to go from 0% to 100% -> 100ms ex. 100/0.1 = 1000%/s*)
		SendCaliResultToFAT : BOOL;
	END_VAR
	VAR_OUTPUT
		Active : BOOL;
		amplitude_out : REAL;
		frequency_out : REAL;
		Braking : BOOL;
		BrakingToAmplitudePct : REAL; (*Amplitude that we are currently braking to "open loop".*)
		HoldPhase : BOOL;
		CalibrateStatus : STRING[60];
		CalibrateDone : BOOL;
		SinePhase : REAL;
		SineOut : REAL;
		SaveConfig : BOOL;
		UpdateFilter : BOOL;
		TestPulses : BOOL;
	END_VAR
	VAR
		VibOptimizerAmplitude_0 : VibOptimizerAmplitude;
		VibOptimizerFrequency_0 : VibOptimizerFrequency;
		LookupTbl_PhaseTarget : LookupTbl;
		LookupTbl_BoostCurrent : LookupTbl;
		LookupTbl_FreqFromCurrent : LookupTbl;
		LookupTbl_CurrentFromPercent : LookupTbl;
		paramsBoostCurrentLUT : LUT_typ := (X:=[10,20,30,40,50,60,70,80,90,100,10(0.0)],Y:=[0.45,0.6,0.7425,0.8885,1.0345,1.1805,1.3265,1.4725,1.6185,1.7645,10(0.0)]);
		cali : VibControlCalibration_typ;
		state : UINT;
		frequency : REAL;
		SetAmplitudeLatched : REAL;
		time : REAL;
		sin_ref : REAL;
		old_sin : REAL;
		brakeAmplitude : REAL := 0.9;
		phi : REAL;
		sin_out : REAL;
		phaseShift : REAL;
		sin_abs : REAL;
		phaseShiftLocal : REAL;
		MC_BR_CyclicWrite_0 : MC_BR_CyclicWrite;
		FreqLoopRate : TIME := T#50ms;
		PhaseTarget : REAL := 70;
		lastSetAmplitude : REAL;
		lastSetAmplitudeLatched : REAL;
		brakeTime : REAL := 0.2;
		TestNormal : BOOL;
		PIController_Ampl : PIController;
		PIController_Phase : PIController;
		currentZeroCrossing : BOOL;
		zeroCrossingCount : USINT;
		TestProduction : BOOL;
		TransientAmplitudeKp : REAL := 0.02;
		TransientAmplitudeKi : REAL := 0;
		SteadyAmplitudeKp : REAL := 0.01;
		SteadyAmplitudeKi : REAL := 0.000375;
		SteadyLowAmplitudeKp : REAL := 0.004;
		SteadyLowAmplitudeKi : REAL := 0.00015;
		ErrorLimitTansient : REAL;
		ErrorLimitScaling : REAL := 0.9;
		gainState : INT;
		TON_Transient : TON;
		transientSetAmplitude : REAL;
		count : USINT;
		FeedForwardScaling : REAL := 0.98;
		WaitPeriodsAfterBrake : REAL := 4.0;
		LimitValueToUseNormalKpKi : REAL := 15.0;
		BoostAmplitudeLimit : REAL := 2.0;
		AddToBoostCurrent : REAL;
		measureBoostTime : BOOL;
		ErrorTimeout : BOOL;
		MachineType : USINT;
		TON_ControllerStuck : TON;
		i : USINT;
		DevForce : BOOL;
		TON_running : TON;
		MTBasicsLimiter_0 : MTBasicsLimiter;
		SetAmplitudeChange : REAL;
		oldManualPercent : REAL;
	END_VAR
END_FUNCTION_BLOCK

FUNCTION SkewedGaussianPDF : REAL
	VAR_INPUT
		x : REAL;
		xi : REAL;
		omega : REAL;
		alpha : REAL;
	END_VAR
	VAR
		tempNormPDF : REAL;
		tempNormCDF : REAL;
		a : REAL;
		sign : INT;
		temp : REAL;
		xPDF : REAL;
		xCDF : REAL;
	END_VAR
END_FUNCTION

FUNCTION_BLOCK TimeDelay
	VAR_INPUT
		Enable : BOOL; (*Enables the function block*)
		In : REAL; (*Input signal*)
		Dt : REAL; (*Sampling period [s]*)
		Delay : REAL; (*Delay [s]*)
	END_VAR
	VAR_OUTPUT
		Out : REAL; (*Delayed signal*)
	END_VAR
	VAR
		lastIn : REAL;
	END_VAR
END_FUNCTION_BLOCK

FUNCTION RoundToPrecision : REAL
	VAR_INPUT
		value : REAL;
		precision : INT;
	END_VAR
	VAR
		multiplier : REAL;
	END_VAR
END_FUNCTION

FUNCTION_BLOCK VibOptimizerAmplitude
	VAR_INPUT
		Set : BOOL;
		Get : BOOL;
		Key : REAL; (*Amplitude*)
		Value : REAL; (*Current*)
		VibratorType : USINT;
		paramsCurrentLUT : REFERENCE TO LUT_typ; (*GetCurrentFromAmplitude*)
		Error : REAL;
	END_VAR
	VAR_OUTPUT
		Out : REAL;
	END_VAR
	VAR
		found : BOOL;
		lookup : ARRAY[0..MAX_ELEMENTS] OF lookup_typ;
		i : USINT;
		lastIdx : USINT;
		LookupTbl_Amplitude : LookupTbl;
	END_VAR
END_FUNCTION_BLOCK

FUNCTION GetPhaseDelay : REAL
	VAR_INPUT
		Frequency : REAL;
	END_VAR
	VAR
		w : REAL;
		wc : REAL := 2 * 3.14159 * 150;
		wb : REAL := 2 * 3.14159 * 10;
		A : REAL;
		B : REAL;
		real2 : REAL;
		imag2 : REAL;
	END_VAR
END_FUNCTION

FUNCTION_BLOCK VibOptimizerFrequency
	VAR_INPUT
		Set : BOOL;
		Get : BOOL;
		Reset : BOOL; (*Will reset any saved values.*)
		Key : REAL; (*Amplitude*)
		Value : REAL; (*Current*)
		paramsFrequencyLUT : REFERENCE TO LUT_typ; (*GetFrequencyFromAmplitude*)
		Error : REAL;
	END_VAR
	VAR_OUTPUT
		Out : REAL;
	END_VAR
	VAR
		found : BOOL;
		lookup : ARRAY[0..MAX_ELEMENTS] OF lookup_typ;
		i : USINT;
		lastIdx : USINT;
		LookupTbl_Frequency : LookupTbl;
	END_VAR
END_FUNCTION_BLOCK
```

#### VibFeedback.st
```iecst
FUNCTION_BLOCK VibFeedback

	MC_BR_CyclicRead_0.Enable := Enable;
	MC_BR_CyclicRead_0.Axis := Axis;
	//MC_BR_CyclicRead_0.ParID := 14433;
	//MC_BR_CyclicRead_0.DataType := ncPAR_TYP_REAL;
	MC_BR_CyclicRead_0.DataAddress := ADR(voltage[1]); // voltage[2] = voltage[i-1]
	MC_BR_CyclicRead_0();

	MC_BR_CyclicRead_1.Enable := Enable;
	MC_BR_CyclicRead_1.Axis := Axis;
	//MC_BR_CyclicRead_1.ParID := 14425;
	//MC_BR_CyclicRead_1.DataType := ncPAR_TYP_REAL;
	MC_BR_CyclicRead_1.DataAddress := ADR(voltage[2]); // voltage[3] = voltage[i]
	MC_BR_CyclicRead_1();

	MC_BR_CyclicRead_2.Enable := Enable;
	MC_BR_CyclicRead_2.Axis := Axis;
	//MC_BR_CyclicRead_2.ParID := 14435;
	//MC_BR_CyclicRead_2.DataType := ncPAR_TYP_REAL;
	MC_BR_CyclicRead_2.DataAddress := ADR(current[1]); // current[2] = current[i-1]
	MC_BR_CyclicRead_2();

	MC_BR_CyclicRead_3.Enable := Enable;
	MC_BR_CyclicRead_3.Axis := Axis;
	//MC_BR_CyclicRead_3.ParID := 14427;
	//MC_BR_CyclicRead_3.DataType := ncPAR_TYP_REAL;
	MC_BR_CyclicRead_3.DataAddress := ADR(current[2]); // current[3] = current[i]
	MC_BR_CyclicRead_3();

	// Go to 0 and update filters if we get Update command
	IF UpdateFilter AND NOT oldUpdateFilter THEN
		state := 0;
	END_IF
	oldUpdateFilter := UpdateFilter;

	TON_PhaseValid.IN := Amplitude_out > 0.0;
	TON_PhaseValid();

	FOR i:=1 TO 2 DO

		CASE state OF
			0:

				IF Enable THEN
					// Setup FBs.
					MTFilterBandPass_3rdHarmonic.Enable := TRUE;
					MTFilterBandPass_3rdHarmonic.CenterFrequency := config.centerFrequencyBPF;
					MTFilterBandPass_3rdHarmonic.Bandwidth := SEL(MachineSize=0,2.5,10.0);
					MTFilterBandPass_3rdHarmonic.Order := 2;
					MTFilterBandPass_3rdHarmonic.Type := mtFILTER_BUTTERWORTH;

					MTFilterLowPass_Amplitude.Enable := TRUE;
					MTFilterLowPass_Amplitude.Order := 2;
					MTFilterLowPass_Amplitude.CutOffFrequency := 300;

					MTFilterLowPass_Phase.Enable := TRUE;
					MTFilterLowPass_Phase.Order := 2;
					MTFilterLowPass_Phase.CutOffFrequency := 300;

					TON_PhaseValid.PT := SEL(MachineSize=0,T#150ms,T#100ms);
					hammingLength := SEL(MachineSize=0,100,50); // 50 for small CF, 100 for big CF

					// Create hamming window
					FOR j:=0 TO MAX_SAMPLES_GOERTZEL DO
						hammingWindow[j] := getHammingWindow(MAX_SAMPLES_GOERTZEL,j);
					END_FOR

					IF UpdateFilter THEN
						state := 5;
					ELSE
						state := 10;
					END_IF
				END_IF

			5:
				MTFilterBandPass_3rdHarmonic.Update := TRUE;
				MTFilterBandPass_3rdHarmonic();

				UpdateFilterDone := MTFilterBandPass_3rdHarmonic.UpdateDone;

				IF NOT UpdateFilter THEN
					UpdateFilterDone := FALSE;
					MTFilterBandPass_3rdHarmonic.Update := FALSE;
					MTFilterBandPass_3rdHarmonic();
					state := 10;
				END_IF

			10:

				IF Amplitude_out > 0.0 THEN
					time := time + dt; // Because it is a for-loop it will run in 400us
					timeHalfPeriod := (1/Frequency)*0.5;
					voltageZeroCrossing := (voltage[i-1] <= 0 AND voltage[i] > 0) OR (voltage[i-1] >= 0 AND voltage[i] < 0);
				END_IF

				IF time >= timeHalfPeriod AND voltageZeroCrossing THEN
					time := 0;
					IF Amplitude_out > 0.0 THEN
						hammingIdx := 0;
						AmplitudeCurrent := SEL(Amplitude_out > 0.0,0.01,Amplitude_out); // SEL to avoid division by 0

						LookupTbl_Percent.Enable := TRUE;
						LookupTbl_Percent.X := ADR(config.lookUpPercentFromAmplitude.X);
						LookupTbl_Percent.Y := ADR(config.lookUpPercentFromAmplitude.Y);
						LookupTbl_Percent();

						goertzelCount := 0;

						state := 20;
					END_IF
				ELSE
					MTFilterBandPass_3rdHarmonic.In := 0;
					MTFilterBandPass_3rdHarmonic();
					MTFilterLowPass_Amplitude.In := 0;
					MTFilterLowPass_Amplitude();
					MTFilterLowPass_Phase.In := 90;
					MTFilterLowPass_Phase();
				END_IF

//			15:
//
//				MTFilterBandPass_3rdHarmonic.In := (voltage[i]);
//				IF hammingIdx < hammingLength/2 THEN
//					MTFilterBandPass_3rdHarmonic.In := MTFilterBandPass_3rdHarmonic.In * HammingWindow(hammingIdx, hammingLength);
//					hammingIdx := hammingIdx + 1;
//				END_IF
//				MTFilterBandPass_3rdHarmonic();
//				Feedback := MTFilterBandPass_3rdHarmonic.Out/AmplitudeCurrent;
//
//				IF (current[i-1] >= 0 AND current[i] < 0) OR (current[i-1] <= 0 AND current[i] > 0) THEN
//					state := 20;
//				END_IF

			20:
				IF Braking THEN
					time := 0;
					Amplitude := BrakingToAmplitudePct;
					MTFilterBandPass_3rdHarmonic.In := 0.0; // Prime with 0 because we start again after brake at zero-crossing
					MTFilterBandPass_3rdHarmonic();
					MTFilterLowPass_Amplitude.In := BrakingToAmplitudePct; // Prime with the amplitude (in percent) we are braking to open-loop.
					MTFilterLowPass_Amplitude();

					state := 30;
				ELSIF Amplitude_out > 0.0 THEN

					MTFilterBandPass_3rdHarmonic.In := voltage[i];
					IF hammingIdx < hammingLength/2 THEN
						MTFilterBandPass_3rdHarmonic.In := MTFilterBandPass_3rdHarmonic.In * HammingWindow(hammingIdx, hammingLength);
						hammingIdx := hammingIdx + 1;
					END_IF
					MTFilterBandPass_3rdHarmonic();
					Feedback := MTFilterBandPass_3rdHarmonic.Out/AmplitudeCurrent;

					IF ABS(Feedback) > peakVib THEN
						peakVib := ABS(Feedback);
					END_IF

					IF ABS(current[i]) > peakCurr THEN
						peakCurr := ABS(current[i]);
					END_IF

					// Detect zero-crossings on current.
					IF (current[i-1] >= 0 AND current[i] < 0) THEN
						LookupTbl_Percent.In := peakVib;
						LookupTbl_Percent();

						MTFilterLowPass_Amplitude.In := SEL(Calibrating,LookupTbl_Percent.Out,peakVib);  // If calibrating use peakVib directly (the LUT is being updated by VibControl)
						MTFilterLowPass_Amplitude();
						Amplitude := MTFilterLowPass_Amplitude.Out;
						AmplitudeRaw := peakVib;
						AmplitudeCurrent := SEL(peakCurr > 0.0,0.01,peakCurr); // SEL to avoid division by 0
						AmplitudeValid := TRUE;

						peakVib := 0;
						peakCurr := 0;
					END_IF

//					IF (lastBPF >= 0 AND Feedback < 0) AND lastSinePhase < SinePhase AND NOT HoldPhase THEN
//						feedbackInterpolation := (((-lastBPF)/(Feedback-lastBPF))+(i-1))/2.0;
//						IF SinePhase < 2.0*PI/3.0 THEN
//							MTFilterLowPass_Phase.In := lastSinePhase + (SinePhase-lastSinePhase)*feedbackInterpolation;
//							MTFilterLowPass_Phase.In := ((MTFilterLowPass_Phase.In / 2.0*PI/3.0) * 180) - SEL(Braking, 0, 90);
//							MTFilterLowPass_Phase();
//							Phase := MTFilterLowPass_Phase.Out;
//							PhaseValid := TRUE;
//						END_IF
//					END_IF

					IF goertzelCount <= MAX_SAMPLES_GOERTZEL THEN
						samples[goertzelCount] := voltage[i];
						samplesCurr[goertzelCount] := current[i];
						goertzelCount := goertzelCount+1;
					ELSIF current[i-1] <= 0.0 AND current[i] > 0.0 THEN
						goertzelMagPhase_0.samples := ADR(samples);
						goertzelMagPhase_0.window := ADR(hammingWindow);
						goertzelMagPhase_0.frequency := (Frequency)*3;
						goertzelMagPhase_0.sampleRate := 2500;
						goertzelMagPhase_0();
						phase[0] := goertzelMagPhase_0.phase;
						goertzelMagPhase_1.samples := ADR(samples);
						goertzelMagPhase_1.window := ADR(hammingWindow);
						goertzelMagPhase_1.frequency := Frequency;
						goertzelMagPhase_1.sampleRate := 2500;
						goertzelMagPhase_1();
						phase[1] := goertzelMagPhase_0.phase;
						goertzelMagPhase_2.samples := ADR(samplesCurr);
						goertzelMagPhase_2.window := ADR(hammingWindow);
						goertzelMagPhase_2.frequency := (Frequency)*3;
						goertzelMagPhase_2.sampleRate := 2500;
						goertzelMagPhase_2();
						phase[2] := goertzelMagPhase_0.phase;
						goertzelMagPhase_3.samples := ADR(samplesCurr);
						goertzelMagPhase_3.window := ADR(hammingWindow);
						goertzelMagPhase_3.frequency := Frequency;
						goertzelMagPhase_3.sampleRate := 2500;
						goertzelMagPhase_3();
						phase[3] := goertzelMagPhase_0.phase;
						oldGoertzelPhaseStart := goertzelPhaseStart;
						goertzelCount := 0;
						goertzelRef := fmod((goertzelMagPhase_3.phase+PI)*3, 2*PI);
						goertzelSignal := goertzelMagPhase_0.phase+PI;
						goertzelPhase := (goertzelRef - goertzelSignal) * 180.0/PI;

						IF NOT HoldPhase THEN
							Phase := goertzelPhase;
							PhaseValid := TON_PhaseValid.Q;
						END_IF

						//						goertzelPhase := (goertzelMagPhase_3.phase-goertzelMagPhase_0.phase/3) * 180.0/PI;
						//						IF goertzelPhase <= -120 THEN
						//							goertzelPhase := (goertzelPhase + 240.0) / 120.0 * 360.0;
						//						ELSIF goertzelPhase <= 0 THEN
						//							goertzelPhase := (goertzelPhase + 120.0) / 120.0 * 360.0;
						//						ELSIF goertzelPhase <= 120 THEN
						//							goertzelPhase := (goertzelPhase) / 120.0 * 360.0;
						//						ELSE
						//							goertzelPhase := (goertzelPhase - 120.0) / 120.0 * 360.0;
						//						END_IF

						goertzelPhaseComp := goertzelPhase-goertzelPhaseStart*goertzelScaling;
						goertzelPhaseStart := SinePhase;

						// Goertzel amplitude
						AmplitudeGoertzel := goertzelMagPhase_0.magnitude/AmplitudeCurrent;
					END_IF

					// last:
					lastBPF := Feedback;
				ELSE
					LookupTbl_Percent.In := 0;
					LookupTbl_Percent();
					LookupTbl_Percent.Enable := FALSE;
					LookupTbl_Percent();
					peakVib := 0;
					Amplitude := 0;
					AmplitudeGoertzel := 0;
					AmplitudeRaw := 0;
					Phase := 0;
					PhaseGoertzel := 0;
					cnt := 0;
					lastBPF := 0;
					time := 0;
					PhaseValid := FALSE;
					AmplitudeValid := FALSE;

					ActAmplitudeGoertzel := 0;
					state := 10;
				END_IF

			30:

				IF NOT Braking THEN
					time := time + dt;
					timeHalfPeriod := (1/Frequency)*0.5;
					voltageZeroCrossing := (voltage[i-1] <= 0 AND voltage[i] > 0) OR (voltage[i-1] >= 0 AND voltage[i] < 0);

					IF time >= timeHalfPeriod AND voltageZeroCrossing THEN
						goertzelCount := 0;
						peakVib := 0;
						time := 0;
						peakCurr := Amplitude_out; // amplitude_out was much bigger when brake started - therefore set amplitude_out to the setpoint we use now. That will be much closer to the actual current amplitude.
						state := 20;
					END_IF
				END_IF
				MTFilterBandPass_3rdHarmonic.In := 0.0;
				MTFilterBandPass_3rdHarmonic();
				MTFilterLowPass_Amplitude.In := BrakingToAmplitudePct; // Prime with the amplitude (in percent) we are braking to open-loop.
				MTFilterLowPass_Amplitude();

		END_CASE

	END_FOR

	lastSinePhase := SinePhase;

	// Calc phase with accelerometer using 800us: (only for testing!!)
	IF Calibrating OR testPhaseUsingAcc THEN
		IF (lastCurrAcc <= 0 AND SineOut > 0) THEN
			tmpTimeAcc := (-lastCurrAcc*0.0008)/(SineOut-lastCurrAcc);  						// Calculate the time of zero crossing
			cntAcc := 0;
			CalcPhasePosAcc := TRUE;
		END_IF

		IF CalcPhasePosAcc THEN

			IF (lastRawVib <= 0 AND RawVib > 0) AND cntAcc > 1 THEN
				tmpTimeAirgap := ((-lastRawVib*0.0008)/(RawVib-lastRawVib));
				PhaseAcc := (cntAcc*0.0008 + tmpTimeAirgap + (0.0008 - lastTmpTimeAcc)) / (1.0/(Frequency * 2.0)) * 180.0;
				CalcPhasePosAcc := FALSE;
			END_IF
			cntAcc := cntAcc + 1;
		END_IF
	END_IF

	// Save last
	voltage[0] := voltage[2];
	current[0] := current[2];
	lastRawVib := RawVib;
	lastTmpTimeAcc := tmpTimeAcc;
	lastCurrAcc := SineOut;
END_FUNCTION_BLOCK

FUNCTION_BLOCK VibFeedbackOld

	CASE state OF
		0:
			IF Enable THEN
				currentLPF[0] := 0;
				voltageLPF[0] := 0;
				IF Simulation THEN
					state := 100;
				ELSE
					state := 10;
				END_IF
			END_IF

		10:
//
//			MC_BR_CyclicRead_2.Enable := TRUE;
//			MC_BR_CyclicRead_2.Axis := Axis;
//			MC_BR_CyclicRead_2.ParID := 14433;
//			MC_BR_CyclicRead_2.DataType := ncPAR_TYP_REAL;
//			MC_BR_CyclicRead_2.DataAddress := ADR(voltage[1]); // voltage[2] = voltage[i-1]
//			MC_BR_CyclicRead_2();
//
//			MC_BR_CyclicRead_3.Enable := TRUE;
//			MC_BR_CyclicRead_3.Axis := Axis;
//			MC_BR_CyclicRead_3.ParID := 14425;
//			MC_BR_CyclicRead_3.DataType := ncPAR_TYP_REAL;
//			MC_BR_CyclicRead_3.DataAddress := ADR(voltage[2]); // voltage[3] = voltage[i]
//			MC_BR_CyclicRead_3();
//
//			MC_BR_CyclicRead_6.Enable := TRUE;
//			MC_BR_CyclicRead_6.Axis := Axis;
//			MC_BR_CyclicRead_6.ParID := 14435;
//			MC_BR_CyclicRead_6.DataType := ncPAR_TYP_REAL;
//			MC_BR_CyclicRead_6.DataAddress := ADR(current[1]); // current[2] = current[i-1]
//			MC_BR_CyclicRead_6();
//
//			MC_BR_CyclicRead_7.Enable := TRUE;
//			MC_BR_CyclicRead_7.Axis := Axis;
//			MC_BR_CyclicRead_7.ParID := 14427;
//			MC_BR_CyclicRead_7.DataType := ncPAR_TYP_REAL;
//			MC_BR_CyclicRead_7.DataAddress := ADR(current[2]); // current[3] = current[i]
//			MC_BR_CyclicRead_7();
//
//			MC_BR_CyclicReadDataInfo_0.Enable := TRUE;
//			MC_BR_CyclicReadDataInfo_0.Axis := Axis;
//			MC_BR_CyclicReadDataInfo_0();

			FOR i:=1 TO 2 DO
				// Generating the LPF current and voltage of the subsampled current and voltage from the drive
				MTFilterLowPass_0.Enable := TRUE;
				MTFilterLowPass_0.Order := 4;
				MTFilterLowPass_0.CutOffFrequency := CutOffFrequency;
				MTFilterLowPass_0.In := current[i];
				MTFilterLowPass_0();

				MTFilterLowPass_1.Enable := TRUE;
				MTFilterLowPass_1.Order := 4;
				MTFilterLowPass_1.CutOffFrequency := CutOffFrequency;
				MTFilterLowPass_1.In := voltage[i];
				MTFilterLowPass_1();

				currentLPF[i] := MTFilterLowPass_0.Out;

				TimeDelay_0.Enable := TRUE;
				TimeDelay_0.Dt := 0.0004;
				TimeDelay_0.In := MTFilterLowPass_1.Out;
				TimeDelay_0.Delay := TimeDelayVoltage;
				TimeDelay_0();
				voltageLPF[i] := TimeDelay_0.Out;

			END_FOR

			TON_RunDelay.IN := RunCalculation;
			TON_RunDelay.PT := RunDelay;
			TON_RunDelay();

			IF NOT TON_RunDelay.Q THEN
				Amplitude := 0;
				AmplitudeFast := 0;
				Phase := 0;
				PhaseHMI := 0;
				IF NOT MTFilterBandPass_Airgap.Enable THEN
					MTFilterBandPass_Airgap.CenterFrequency := 50;
					MTFilterBandPass_Airgap.Bandwidth := 30;
					MTFilterBandPass_Airgap.Order := 1;
				END_IF
				MTFilterBandPass_Airgap.Enable := TRUE;
				MTFilterBandPass_Airgap.In := meanAirgap;
				MTFilterBandPass_Airgap();
				IF NOT MTFilterBandPass_AirgapFast.Enable THEN
					MTFilterBandPass_AirgapFast.CenterFrequency := 50;
					MTFilterBandPass_AirgapFast.Bandwidth := 30;
					MTFilterBandPass_AirgapFast.Order := 1;
				END_IF
				MTFilterBandPass_AirgapFast.Enable := TRUE;
				MTFilterBandPass_AirgapFast.In := meanAirgap;
				MTFilterBandPass_AirgapFast();
			END_IF

			TON_CalcDelay.IN := RunCalculation;
			TON_CalcDelay.PT := CalcDelay;
			TON_CalcDelay();

			IF RunCalculation THEN
				FOR i:=1 TO 2 DO
					// If zero crossing of the the current has occured (rising or falling)
					IF (currentLPF[i-1] <= 0 AND currentLPF[i] > 0) OR (currentLPF[i-1] >= 0 AND currentLPF[i] < 0) THEN
						// Calculation of the complete commulative integral to the point at zero crossing
						tmpTime := (-currentLPF[i-1]*dt)/(currentLPF[i]-currentLPF[i-1]);  						// Calculate the time of zero crossing
						a := (voltageLPF[i]-voltageLPF[i-1])/dt;					  							// Calculate voltage slope
						zeroVolt := a*tmpTime+voltageLPF[i-1];						  								// Calculate the voltage at zero crossing
						intCurr[i] := intCurr[i-1] + (0.5*(0+currentLPF[i-1])*(tmpTime)); 		  					// Calculate the instantenous integration of the current at zero crossing
						intVolt[i] := intVolt[i-1] + (0.5*(zeroVolt+voltageLPF[i-1])*(tmpTime));  					// Calculate the instantenous integration of the voltage at zero crossing
						IF intCurr[i] <> 0 THEN
							res := intVolt[i]/intCurr[i];
						ELSE
							res := intVolt[i]/0.00000001;
						END_IF

						voltZeroOffset := intVolt[i] / 2;
						currZeroOffset := intCurr[i] / 2;

						IF TON_RunDelay.Q THEN
							// IMPLEMENTATION OF CONTROL ALGORITHM HERE!
							// Calculate the airgap for half a current wave
							FOR j:=0 TO lastidx-1 DO
								intVoltBuffer[j] := intVoltBuffer[j] - voltZeroOffset;
								intCurrBuffer[j] := intCurrBuffer[j] - currZeroOffset;
								intEMF[j]		:= intVoltBuffer[j]-(res*intCurrBuffer[j]);

								IF intEMF[j] <> 0 THEN
									tmpAirgap := currentLPFBuffer[j] / intEMF[j] ; // Airgap
								ELSE
									tmpAirgap := currentLPFBuffer[j] / 0.00000001;
								END_IF

								tmpAirgap := LIMIT(-1000, tmpAirgap, 1000);

								MTFilterBandPass_Airgap.Enable := TRUE;
								MTFilterBandPass_Airgap.In := tmpAirgap;
								MTFilterBandPass_Airgap();

								MTFilterBandPass_AirgapFast.Enable := TRUE;
								MTFilterBandPass_AirgapFast.In := tmpAirgap;
								MTFilterBandPass_AirgapFast();

								IF RawAirgap THEN
									airgap[j] := MTFilterBandPass_AirgapFast.Out;
								ELSE
									airgap[j] := MTFilterBandPass_Airgap.Out;
								END_IF

							END_FOR

							phaseFound := FALSE;
							FOR j:=1 TO lastidx-1 DO
								IF ABS(airgap[j]) > peakVib THEN
									peakVib := ABS(airgap[j]); // Peak vibration for comparison
								END_IF

								IF (airgap[j-1] >= 0 AND airgap[j] < 0) AND NOT phaseFound THEN // Falling edge
									tmpTimeAirgap := ((-airgap[j-1]*dt)/(airgap[j]-airgap[j-1]));
									lastTmpTimeMinusDt := dt - lastTmpTime;
									phaseCalc := ((j-1)*dt + tmpTimeAirgap + (dt - lastTmpTime)) / (1.0/(Frequency * 2.0)) * 180.0;
									phaseCalc := phaseCalc + PhaseOffset;
									IF phaseCalc > 180 THEN
										phaseCalc := phaseCalc - 180;
									END_IF
									indexJ := j-1;
									phaseFound := TRUE;
								END_IF

							END_FOR

							peak3rdHarmonic := 0.0;
							FOR j:=0 TO idx DO

								IF ABS(voltage3rdHarmonic[j]) > peak3rdHarmonic THEN
									peak3rdHarmonic := ABS(voltage3rdHarmonic[j]);
								END_IF

							END_FOR

							IF NOT MTFilterLowPass_Ampl.Enable THEN
								MTFilterLowPass_Ampl.Enable := TRUE;
								MTFilterLowPass_Ampl.Order := 2;
								MTFilterLowPass_Ampl.CutOffFrequency := 250;
							END_IF
							MTFilterLowPass_Ampl.In := peakVib;
							MTFilterLowPass_Ampl();

							KalmanFilter1D_Ampl.Measurement := peakVib;
							KalmanFilter1D_Ampl();
							IF NOT KalmanFilter1D_Ampl.Enable THEN
								KalmanFilter1D_Ampl.Enable := TRUE;
								KalmanFilter1D_Ampl.KalmanGain := 0.1;
								KalmanFilter1D_Ampl.MeasureVariance := 1;
								KalmanFilter1D_Ampl.ProcessVariance := 0.1;
							END_IF

							IF NOT MTFilterLowPass_Phase.Enable THEN
								MTFilterLowPass_Phase.Enable := TRUE;
								MTFilterLowPass_Phase.Order := 2;
								MTFilterLowPass_Phase.CutOffFrequency := 250;
							END_IF

							IF NOT HoldPhase THEN
								MTFilterLowPass_Phase.In := phaseCalc;
								MTFilterLowPass_Phase();
							END_IF

							IF NOT MTBasicsDT1_ActAmpl.Enable THEN
								MTBasicsDT1_ActAmpl.Gain := 1;
								MTBasicsDT1_ActAmpl.TimeConstant := 1;
							END_IF
							MTBasicsDT1_ActAmpl.Enable := TRUE;
							MTBasicsDT1_ActAmpl.In := MTFilterLowPass_Ampl.Out;
							MTBasicsDT1_ActAmpl();

							IF TON_RunDelay.Q THEN
								Amplitude := RoundToPrecision(MTFilterLowPass_Ampl.Out, 3);
								AmplitudeFast := RoundToPrecision(MTFilterLowPass_Ampl.In, 3);
								Phase := RoundToPrecision(MTFilterLowPass_Phase.Out, 0);
								PhaseFast := RoundToPrecision(MTFilterLowPass_Phase.In, 0);
//								Amplitude := MTFilterLowPass_Ampl.Out;
//								AmplitudeFast := MTFilterLowPass_Ampl.In;
//								Phase := MTFilterLowPass_Phase.Out;
//								PhaseFast := MTFilterLowPass_Phase.In;
								PhaseHMI := Phase;
							END_IF
						END_IF

						// Value for comparison to correct airgap trace in 800�s
						tmpAirgapTrace := lastidx;
						// Reset last array index and Summed airgap
						lastidx    	:= 0;
						peakVib 	:= 0;
						idx := 0;
						// Reset cummulative integrals
						intCurr[i] := (0.5*(currentLPF[i]+0)*(dt-tmpTime)); 						// Reset the cummulative integration of the current
						intVolt[i] := (0.5*(voltageLPF[i]+zeroVolt)*(dt-tmpTime));  						// Reset the cummulative integration of the voltage

						// Put values into buffer and increment the last index
						intVoltBuffer[lastidx] := intVolt[i];
						intCurrBuffer[lastidx] := intCurr[i];
						currentLPFBuffer[lastidx] := currentLPF[i];
						lastidx := lastidx + 1;
						lastTmpTime := tmpTime;
						// IF NO RISING OR FALLING EDGE ON CURRENT
					ELSE
						intCurr[i] := intCurr[i-1] + (0.5*(currentLPF[i]+currentLPF[i-1])*dt);				// Calculate the cummulative integration of the current
						intVolt[i] := intVolt[i-1] + (0.5*(voltageLPF[i]+voltageLPF[i-1])*dt); 			// Calculate the cummulative integration of the voltage
						// Put values into buffer and increment the last index
						intVoltBuffer[lastidx] := intVolt[i];
						intCurrBuffer[lastidx] := intCurr[i];
						currentLPFBuffer[lastidx] := currentLPF[i];

						IF lastidx = tmpAirgapTrace THEN
							airgap1 := airgap[lastidx];
							intCurr1 := intCurrBuffer[lastidx];
							intVolt1 := intVoltBuffer[lastidx];
						ELSIF lastidx < tmpAirgapTrace THEN
							airgap1 := airgap[lastidx];
							airgap2 := airgap[lastidx+1];
							intCurr1 := intCurrBuffer[lastidx];
							intCurr2 := intCurrBuffer[lastidx+1];
							intVolt1 := intVoltBuffer[lastidx];
							intVolt2 := intVoltBuffer[lastidx+1];
						END_IF
						lastidx := lastidx + 1;
					END_IF

					IF NOT MTFilterBandPass_Voltage3rd.Enable THEN
						MTFilterBandPass_Voltage3rd.CenterFrequency := 75;
						MTFilterBandPass_Voltage3rd.Bandwidth := 5;
						MTFilterBandPass_Voltage3rd.Order := 2;
					END_IF
					MTFilterBandPass_Voltage3rd.Enable := TRUE;

					IF SimCurrent > 0.0 THEN
						voltage3rdHarmonic[idx] := MTFilterBandPass_Voltage3rd.Out/SimCurrent;
						idx := LIMIT(0,idx+1,255);
						MTFilterBandPass_Voltage3rd.In := voltage[i];
					ELSE
						MTFilterBandPass_Voltage3rd.In := 0;
					END_IF
					MTFilterBandPass_Voltage3rd();

				END_FOR

				currentLPF[0] := currentLPF[2]; // Save the last value of this data in the first of next call
				voltageLPF[0] := voltageLPF[2]; // Save the last value of this data in the first of next call
				intCurr[0] := intCurr[2]; 		// Save the last value of this data in the first of next call
				intVolt[0] := intVolt[2]; 		// Save the last value of this data in the first of next call
			ELSE
				FOR i:=1 TO 2 DO
					MTFilterBandPass_Voltage3rd.In := voltage[i];
					MTFilterBandPass_Voltage3rd();
				END_FOR
			END_IF

		100:
			// Simulation

			// 10% Current
			// 100% Current
			// 10% Frequency
			// 100% Frequency

			// Calculate amplitude
			simPrc := 10 + (SimCurrent - simCurr10Prc) * (100 - 10) / (simCurr100Prc - simCurr10Prc);
			xi := simResonance + 1 - simPrc*0.02;
			omega := 1 + 0.2*simPrc/10.0;
			alpha := 20;

			IF NOT MTFilterLowPass_Current.Enable THEN
				MTFilterLowPass_Current.CutOffFrequency := 2;
				MTFilterLowPass_Current.Order := 2;
			END_IF
			MTFilterLowPass_Current.Enable := TRUE;
			MTFilterLowPass_Current.In := MAX(0, SkewedGaussianPDF(Frequency, xi, omega, alpha) * (1.2-(100.0-simPrc)/100.0));;
			MTFilterLowPass_Current();

			Amplitude := MTFilterLowPass_Current.Out;

			// Calculate phase
			phaseRes := 0.999546746760729*xi+0.142274*omega+0.02238;

			IF NOT MTFilterLowPass_Frequency.Enable THEN
				MTFilterLowPass_Frequency.CutOffFrequency := 5;
				MTFilterLowPass_Frequency.Order := 2;
			END_IF
			MTFilterLowPass_Frequency.Enable := TRUE;
			IF MTFilterLowPass_Frequency.Out <= phaseRes THEN
				MTFilterLowPass_Frequency.In := 180 / (1 + EXP(-3 * (Frequency - phaseRes)));
			ELSE
				MTFilterLowPass_Frequency.In := 180 / (1 + EXP(-0.5 * (Frequency - phaseRes)));
			END_IF
			MTFilterLowPass_Frequency();

			Phase := MTFilterLowPass_Frequency.Out;

	END_CASE

END_FUNCTION_BLOCK

FUNCTION SkewedGaussianPDF

	xPDF := (x - xi) / omega;
	tempNormPDF := EXP(-xPDF * xPDF / 2.0) / SQRT(2.0 * 3.14159265358979323846); // NormPDF((x - xi) / omega);

	xCDF := alpha * (x - xi) / omega;
	a := 0.147;
	IF x > 0 THEN
		sign := 1;
	ELSIF x < 0 THEN
		sign := -1;
	ELSE
		sign := 0;
	END_IF;
	temp := 1.0 - EXP(-xCDF * xCDF * (4.0 / 3.14159265358979323846 + a * xCDF * xCDF) / (1.0 + a * xCDF * xCDF));
	tempNormCDF := 0.5 * (1.0 + sign * temp); // NormCDF(alpha * (x - xi) / omega);

	SkewedGaussianPDF := 2.0 * tempNormPDF * tempNormCDF;

END_FUNCTION

FUNCTION_BLOCK TimeDelay
	IF Enable THEN
		Out := lastIn + ((In-lastIn)/Dt)*(Dt-Delay);
		lastIn := In;
	ELSE
		Out := In;
	END_IF
END_FUNCTION_BLOCK

FUNCTION_BLOCK KalmanFilter1D

	IF NOT Enable AND Active THEN
		state := 0;
		Active := FALSE;
	END_IF

	CASE state OF
		0:
			IF Enable THEN
				Active := TRUE;
				ErrorEstimate := 1;
				state := 10;
			END_IF

		10:
			// Prediction phase
			Prediction := Estimation;           // For 1D without control input
			ErrorEstimate := ErrorEstimate + ProcessVariance;

			// Update phase
			KalmanGain := ErrorEstimate / (ErrorEstimate + MeasureVariance);
			Estimation := Prediction + KalmanGain * (Measurement - Prediction);
			ErrorEstimate := (1 - KalmanGain) * ErrorEstimate;
	END_CASE

END_FUNCTION_BLOCK

FUNCTION RoundToPrecision

	multiplier := pow(10.0, INT_TO_REAL(precision));
	RoundToPrecision := TRUNC(value * multiplier + 0.5) / multiplier;

END_FUNCTION

FUNCTION GetPercentFromAmplitude

	GetPercentFromAmplitude := 2.4261*Amplitude-0.0494; //R2=0.9981

END_FUNCTION

FUNCTION GetPhaseDelay

	w := 2 * 3.14159 * Frequency;  (* Convert frequency to angular frequency in rad/s *)
	A := wb / (wc * wc);
	B := 1 / (wc * wc);

	real2 := (A * A * w * w * (A * A * w * w - (B * w * w - 1) * (B * w * w - 1))) / ((A * A * w * w + (B * w * w - 1) * (B * w * w - 1)) * (A * A * w * w + (B * w * w - 1) * (B * w * w - 1)));
	imag2 := -(2 * A * A * A * w * w * w * (B * w * w - 1)) / ((A * A * w * w + (B * w * w - 1) * (B * w * w - 1)) * (A * A * w * w + (B * w * w - 1) * (B * w * w - 1)));

	GetPhaseDelay := atan2(imag2, real2) * (180 / 3.14159);

END_FUNCTION

FUNCTION HammingWindow

	HammingWindow := 0.54 - 0.46*COS((2*3.141593*n)/(N-1));

END_FUNCTION
```
